Fanuc KAREL source: NODE_SIZE.kl

PROGRAM T
%NOLOCKGROUP
VAR
 v0 : PATH
 res : INTEGER
BEGIN
 res = NODE_SIZE(v0)
END T
